(* IEC 61131-3 sources: IRIS-Project/LASAL CONTROL SOFTWARE/LasalProject_2025_09_25/Class/Motore_M4, 1 file *)

(* ---- Motore_M4.st ---- *)
(*!
<Class
	Name               = "Motore_M4"
	Revision           = "0.0"
	RealtimeTask       = "false"
	CyclicTask         = "true"
	DefCyclictime      = "100 ms"
	BackgroundTask     = "false"
	Sigmatek           = "false"
	OSInterface        = "false"
	HighPriority       = "false"
	Automatic          = "false"
	UpdateMode         = "Prescan"
	SharedCommandTable = "true"
	Objectsize         = "(720,180)">
	<Channels>
		<Server Name="ClassSvr" Visualized="false" Initialize="false" WriteProtected="true" Retentive="false"/>
		<Server Name="ErrorState" Visualized="false" Initialize="false" WriteProtected="true" Retentive="false"/>
		<Server Name="M4_Correction_Step" Visualized="false" Initialize="false" WriteProtected="false" Retentive="false"/>
		<Server Name="MotoreM4Step" Visualized="false" Initialize="false" WriteProtected="true" Retentive="false"/>
		<Server Name="s_1_3_pelletMode" Visualized="false" Initialize="false" WriteProtected="false" Retentive="false"/>
		<Server Name="s_calibrationMode" Visualized="false" Initialize="false" WriteProtected="false" Retentive="false"/>
		<Server Name="s_DischargeStatus" Visualized="false" Initialize="false" WriteProtected="false" Retentive="false"/>
		<Server Name="s_M4_Homed" Visualized="false" Initialize="false" WriteProtected="false" Retentive="false"/>
		<Server Name="s_measurement_ON" Visualized="false" Initialize="false" WriteProtected="true" Retentive="false"/>
		<Server Name="s_pelletInTrolley" Visualized="false" Initialize="false" WriteProtected="false" Retentive="false"/>
		<Server Name="s_pelletMeasured" Visualized="false" Initialize="false" WriteProtected="false" Retentive="false"/>
		<Server Name="s_target_misurati" Visualized="false" Initialize="false" WriteProtected="false" Retentive="false"/>
		<Client Name="c_MaxCurrent" Required="true" Internal="false"/>
		<Client Name="c_TimerDis" Required="false" Internal="false"/>
		<Client Name="c_TimerMov" Required="true" Internal="false"/>
		<Client Name="Comando_M4" Required="true" Internal="false"/>
		<Client Name="Comando_to_M8Class" Required="true" Internal="false"/>
		<Client Name="M4_LS" Required="false" Internal="false"/>
		<Client Name="SetPositionController" Required="true" Internal="false"/>
	</Channels>
</Class>
*)
Motore_M4 : CLASS
	TYPE
	  t_sequence_Cmd_motore_M4 :  //! <Type Public="true" Name="t_sequence_Cmd_motore_M4"/>
	  (
	    Cmd_motore_M4_idle,
	    Cmd_motore_M4_homing,
	    Cmd_motore_M4_phasing,
	    Cmd_motore_M4_movement,
	    Cmd_motore_M4_reset,
	    Cmd_motore_M4_stop,
	    Cmd_motore_M4_stopped,
	    Cmd_motore_M4_Error,
	    Cmd_motore_M4_movement_2
	  )$UDINT;
	END_TYPE
  //Servers:
	ClassSvr 	: SvrChCmd_DINT;
	MotoreM4Step 	: SvrCh_t_sequence_Cmd_motore_M4_PTofCls_Motore_M4;
	ErrorState 	: SvrCh__LMCAXIS_ERROR;
	s_measurement_ON 	: SvrCh_DINT;
	s_M4_Homed 	: SvrCh_DINT;
	M4_Correction_Step 	: SvrCh_DINT;
	s_target_misurati 	: SvrCh_DINT;
	s_calibrationMode 	: SvrCh_DINT;
	s_1_3_pelletMode 	: SvrCh_DINT;
	s_pelletMeasured 	: SvrCh_DINT;
	s_pelletInTrolley 	: SvrCh_DINT;
	s_DischargeStatus 	: SvrCh_DINT;
  //Clients:
	Comando_M4 	: CltChCmd__LMCAxis;
	Comando_to_M8Class 	: CltChCmd_Motore_M7;
	M4_LS 	: CltCh_DINT;
	c_MaxCurrent 	: CltCh_DINT;
	SetPositionController 	: CltCh_DINT;
	c_TimerDis 	: CltCh_DINT;
	c_TimerMov 	: CltCh_DINT;
  //Variables:
		ActCommand 	: t_sequence_Cmd_motore_M4;
		M4_homed 	: BOOL;
		M4_MovementStep 	: DINT;
		v_MeasurementStartOver 	: BOOL;
		v_DiscahrgeMisure_End 	: BOOL;
		v_M8_inBlockPos 	: BOOL;
		v_ErrorState 	: DINT;
		HomingStep 	: DINT;
		Movement_step 	: DINT;
		v_StartHomingCase 	: DINT;
		v_StartMovementCase 	: DINT;
		v_offset_Dis 	: DINT;
		v_target_misurati 	: DINT;
		v_M4_LS 	: DINT;
		v_ACK_M4_Mov 	: DINT;
		flag 	: DINT;
		v_startTimer 	: BOOL;
		v_pelletMeasured 	: DINT;
		v_pelletInTrolley 	: DINT;
		v_PelletAvailable 	: DINT;
  //Functions:

	FUNCTION VIRTUAL GLOBAL Init;

	FUNCTION VIRTUAL GLOBAL CyWork
		VAR_INPUT
			EAX 	: UDINT;
		END_VAR
		VAR_OUTPUT
			state (EAX) 	: UDINT;
		END_VAR;

	FUNCTION GLOBAL SetSequenceState
		VAR_INPUT
			Cmd_motore 	: t_sequence_Cmd_motore_M4;
			Motion_Type 	: DINT;
			StartCase 	: DINT;
		END_VAR
		VAR_OUTPUT
			retcode 	: DINT;
		END_VAR;

	FUNCTION GLOBAL GetHomedState
		VAR_OUTPUT
			Homed 	: BOOL;
		END_VAR;

	FUNCTION GLOBAL GetMisurationStartOver
		VAR_INPUT
			Status 	: BOOL;
		END_VAR;

	FUNCTION GLOBAL SetDischargeOver
		VAR_OUTPUT
			Status 	: BOOL;
		END_VAR;

	FUNCTION GLOBAL GetM8Status
		VAR_INPUT
			Status 	: BOOL;
		END_VAR
		VAR_OUTPUT
			retcode 	: DINT;
		END_VAR;

	FUNCTION GLOBAL GetErrorState
		VAR_OUTPUT
			ErrorState 	: DINT;
		END_VAR;

	FUNCTION GLOBAL GetMoveDone
		VAR_OUTPUT
			OutParam 	: DINT;
		END_VAR;

	FUNCTION GLOBAL GetPelletAvailable
		VAR_INPUT
			Param 	: DINT;
		END_VAR;
  //Tables:
	FUNCTION @STD
		VAR_OUTPUT
			ret_code	: CONFSTATES;
		END_VAR;
	FUNCTION GLOBAL TAB @CT_;
END_CLASS;

#pragma usingLtd _LMCAxis
#pragma usingLtd Motore_M7

FUNCTION VIRTUAL GLOBAL Motore_M4::CyWork
	VAR_INPUT
		EAX 	: UDINT;
	END_VAR
	VAR_OUTPUT
		state (EAX) 	: UDINT;
	END_VAR

  v_M4_LS:=M4_LS.Read();
  s_M4_Homed.Write(input:=M4_homed);

  s_target_misurati.Write(input:=v_target_misurati);

  case MotoreM4Step of
//===========================================================================================

    Cmd_motore_M4_idle:

    if Comando_M4.AxisError.HwError then
      v_ErrorState:=1;   ;
      MotoreM4Step:=Cmd_motore_M4_Error;
    end_if;
    v_ACK_M4_Mov:=0;
//===========================================================================================

    Cmd_motore_M4_homing:
    //lo muovo fino al click dello switch, questa posizione corrisponde a quella in cui un target, se nello slider, cade nella posizione di carico
    if Comando_M4.AxisError.HwError then
      v_ErrorState:=1;
      HomingStep:=0;
      MotoreM4Step:=Cmd_motore_M4_Error;
    end_if;

    case HomingStep of

    0://idle
      HomingStep:=v_StartHomingCase;

    5:
      if v_M4_LS then //Motore già in posizione.
        HomingStep:=50;
      else
        HomingStep:=10;
      end_if;

    10://POWER ON

      if (Comando_M4.AxisStatus.PowerOn=0) & (Comando_M4.AxisStatus.ReadyToPowerOn) then
        Comando_M4.PowerOn(Mode:=_LMCAXIS_MOVEDIRECTION::LMCAXIS_MOVE_ANY_WAY);
      elsif Comando_M4.AxisStatus.PowerOn then
        HomingStep:=20;
      end_if;

    20:

      Comando_M4.TuneAxis(Position:=P_M4_H, Speed:=V_M4, Accel:=A_M4, Mode:=LMCAXIS_TUNE_POSITON_IN_POSITIVE_DIRECTION, WaitTime:=0, Jerk:=J_M4);
      HomingStep:=30;

    30:
      if v_M4_LS=0 then //quando tocca LS
        Comando_M4.StopMove(Decel:=A_M4, Jerk:=J_M4);
        HomingStep:=40;
      end_if;

    40://Controllo che il motore si sia fermato

      if Comando_M4.AxisStatus.Standstill then
          Comando_M4.PowerOff(Mode:=LMCAXIS_IMMEDIATE_STOPP);
          HomingStep:=50;
      end_if;

    50:
       if Comando_M4.AxisStatus.PowerOn=0 then
          SetPositionController.Write(input:=0);
          M4_homed:=TRUE;
          MotoreM4Step:=Cmd_motore_M4_idle;
          v_StartHomingCase:=0;
       end_if;

    end_case;

//==================================================================================
     Cmd_motore_M4_movement:

    //
    //BLOCCO DI COMANDI PER MOVIMENTAZIONE MOTORE M4
    //
    //SI TROVA GIA' NELLA POSIZIONE IN CUI PUO' UN TARGET CADE

    if Comando_M4.AxisError.HwError then
      v_ErrorState:=1;
      Movement_step:=0;
      MotoreM4Step:=Cmd_motore_M4_Error;
    end_if;

    case Movement_step of

    0: //IDLE, ATTESA COMANDI| Il motore è già nella posizione di carica->tocca il LS
        Movement_step:=v_StartMovementCase;
    10://M2 si trova nella posizione corretta di caricamento DEVE RUOTARE NEL VERSO CORRETTO PER SCARICARE TARGET, compirà 1 giro completo (quasi)

     if (Comando_M4.AxisStatus.PowerOn=0) & (Comando_M4.AxisStatus.ReadyToPowerOn) then
        Comando_M4.PowerOn(Mode:=LMCAXIS_MOVE_ANY_WAY);
     elsif Comando_M4.AxisStatus.PowerOn then
        Movement_step:=20;
        s_DischargeStatus.Write(input:=0);
     end_if;

    20:

      if v_M8_inBlockPos then
        Movement_Step:=30;
      elsif v_M8_inBlockPos=FALSE then
        Comando_to_M8Class.SetSequenceState(Cmd_motore:=Motore_M7::Cmd_motore_M7_movement, Motion_type:=0, StartCase:=10);//dico al motore di andare in posizione di blocco
        Movement_Step:=25;
      end_if;

    25:
      if v_M8_inBlockPos=true then
        Movement_Step:=30;
        flag:=1;
      end_if;

    30:
      Comando_M4.MoveAbsolute(Position:=(P1_M4+v_offset_Dis), Speed:=V_M4, Accel:=A_M4, Decel:=A_M4, Jerk:=J_M4);
      Movement_Step:=40;

    40:
      IF Comando_M4.InPosition(Mode:=LMCAXIS_NO_POSITIONWINDOW, PositionWindow:=0) & Comando_M4.AxisStatus.Standstill  & v_MeasurementStartOver THEN //se ho scaricato target e dico che è pronto per la misurazione
      //FASE DI MISURAZIONE
        v_pelletMeasured+=1;
        s_pelletMeasured.Write(input:=v_pelletMeasured);
        c_TimerDis.Write(input:=1);
        c_TimerMov.Write(input:=0);
        s_measurement_ON.Write(input:=1);//MISURAZIONE ATTIVA
        s_DischargeStatus.Write(input:=1);
        v_target_misurati+=1;
        Movement_step:=50;
      END_IF;

    50:
      if v_MeasurementStartOver=FALSE then
        v_pelletMeasured+=1;
        s_pelletMeasured.Write(input:=v_pelletMeasured);
        c_TimerDis.Write(input:=0);
        Comando_to_M8Class.SetSequenceState(Cmd_motore:=Motore_M7::Cmd_motore_M7_movement, Motion_type:=1,StartCase:=10);//dico al motore di USCIRE dalla posizione di blocco
        v_target_misurati+=1;
        v_pelletInTrolley+=1;
        s_pelletInTrolley.Write(input:=v_pelletInTrolley);
        s_measurement_ON.Write(input:=0);
        v_offset_Dis+=1200000;

        if s_1_3_pelletMode.Read()=1 then
          Movement_Step:=80;
        elsif s_1_3_pelletMode.Read()=0 then
          Movement_Step:=60;
        end_if;

      end_if;

    60:
      if v_target_misurati<6 & Comando_to_M8Class.GetCoupledState()=FALSE then
        Movement_Step:=20;
      elsif v_target_misurati=6 & Comando_to_M8Class.GetCoupledState()=FALSE then
        Comando_M4.PowerOff(Mode:=LMCAXIS_IMMEDIATE_STOPP);
        Movement_Step:=70;
      end_if;

    70:
    if Comando_M4.AxisStatus.PowerOn=0 then
       s_DischargeStatus.Write(input:=2);
       v_DiscahrgeMisure_End:=TRUE;
       Movement_Step:=0;
       MotoreM4Step:=Cmd_motore_M4_idle;
    end_if;

    //Calibration Mode
    80:
      if Comando_to_M8Class.GetCoupledState()=FALSE & Comando_M4.AxisStatus.Standstill then
          Comando_M4.PowerOff(Mode:=LMCAXIS_IMMEDIATE_STOPP);
          Movement_Step:=70;
      end_if;

    end_case;
//========================================================================

    Cmd_motore_M4_movement_2:
    if Comando_M4.AxisError.HwError then
      v_ErrorState:=1;
      Movement_step:=0;
      MotoreM4Step:=Cmd_motore_M4_Error;
    end_if;

    case Movement_step of

    0: //IDLE, ATTESA COMANDI| Il motore è già nella posizione di carica->tocca il LS
        Movement_step:=v_StartMovementCase;
    10://M2 si trova nella posizione corretta di caricamento DEVE RUOTARE NEL VERSO CORRETTO PER SCARICARE TARGET, compirà 1 giro completo (quasi)

     if (Comando_M4.AxisStatus.PowerOn=0) & (Comando_M4.AxisStatus.ReadyToPowerOn) then
        Comando_M4.PowerOn(Mode:=LMCAXIS_MOVE_ANY_WAY);
     elsif Comando_M4.AxisStatus.PowerOn then
        Movement_step:=20;
     end_if;

    20:

      Comando_M4.MoveRelative(Position:=900000, Mode:=LMCAXIS_MOVE_RELATIVE_TO_POSITION , Speed:=V_M4, Accel:=A_M4, Decel:=A_M4, Jerk:=J_M4);
      Movement_step:=30;

    30:

      if Comando_M4.AxisStatus.InPosition then
        v_ACK_M4_Mov:=1;
        Movement_step:=40;
        Comando_M4.PowerOff(Mode:=LMCAXIS_IMMEDIATE_STOPP);
      end_if;

    40:
      Movement_Step:=0;
      v_StartMovementCase:=0;
      MotoreM4Step:=Cmd_motore_M4_idle;

    end_case;
//========================================================================

     Cmd_motore_M4_Error:

      ErrorState:=Comando_M4.AxisError; //AGGIORNAMENTO SERVER
      MotoreM4Step:=Cmd_motore_M4_stop;

//========================================================================
    Cmd_motore_M4_stop:

      if Comando_M4.AxisStatus.Standstill & Comando_M4.AxisStatus.PowerOn=0 then
        MotoreM4Step:=Cmd_motore_M4_stopped;
      else
        Comando_M4.QuickStop(Decel:=1000000);//se asse in errore non esegue neppure l'operazione perchè spento (e in errore)
        Comando_M4.PowerOff(Mode:=LMCAXIS_IMMEDIATE_STOPP);
      end_if;

//========================================================================
    Cmd_motore_M4_stopped:
    //ATTESA RESET

//========================================================================
    Cmd_motore_M4_reset:
      Comando_M4.QuitError();
      Comando_to_M8Class.SetSequenceState(Cmd_motore:=Motore_M7::Cmd_motore_M7_reset, Motion_type:=3, StartCase:=0);
      M4_homed:=FALSE;
      v_ErrorState:=0;
      if Comando_M4.AxisStatus.FiltRdy then
        MotoreM4Step:=Cmd_motore_M4_idle;
      end_if;

      v_MeasurementStartOver:=FALSE;
      v_DiscahrgeMisure_End:=FALSE;
      v_M8_inBlockPos:=0;
      v_offset_Dis:=0;
      v_target_misurati:=0;
      HomingStep:=0;
      Movement_step:=0;
      v_StartHomingCase:=0;
      v_StartMovementCase:=0;
      flag:=0;
      v_ACK_M4_Mov:=0;
      v_M4_LS:=0;
      v_ErrorState:=0;
      v_startTimer:=FALSE;
      s_calibrationMode.Write(input:=0);
      //s_1_3_pelletMode.Write(input:=0);
      s_DischargeStatus.Write(input:=0);

      if v_pelletMeasured/2>=v_PelletAvailable then
          v_pelletMeasured:=0;
          s_pelletMeasured.Write(input:=0);
          v_pelletInTrolley:=0;
          s_pelletInTrolley.Write(input:=0);
      end_if;

//========================================================================

  end_case;

	state := READY;
END_FUNCTION

FUNCTION GLOBAL Motore_M4::SetSequenceState
	VAR_INPUT
		Cmd_motore 	: t_sequence_Cmd_motore_M4;
		Motion_Type 	: DINT;
		StartCase 	: DINT;
	END_VAR
	VAR_OUTPUT
		retcode 	: DINT;
	END_VAR

  if Cmd_motore=Cmd_motore_M4_homing then
    v_StartHomingCase:=StartCase;
  elsif Cmd_motore=Cmd_motore_M4_movement then
    v_StartMovementCase:=StartCase;
  elsif Cmd_motore=Cmd_motore_M4_movement_2 then
    v_StartMovementCase:=StartCase;
  end_if;

  MotoreM4Step:=Cmd_motore;
  retcode:=true;
END_FUNCTION

FUNCTION VIRTUAL GLOBAL Motore_M4::Init
M4_homed:=FALSE;
v_MeasurementStartOver:=FALSE;
v_DiscahrgeMisure_End:=FALSE;
v_M8_inBlockPos:=0;

v_offset_Dis:=0;
v_target_misurati:=0;

HomingStep:=0;
Movement_step:=0;

v_StartHomingCase:=0;
v_StartMovementCase:=0;

flag:=0;

v_ACK_M4_Mov:=0;

v_M4_LS:=0;

v_ErrorState:=0;

v_startTimer:=FALSE;

v_pelletMeasured:=0;
v_pelletInTrolley:=0;

v_PelletAvailable:=0;

END_FUNCTION

FUNCTION GLOBAL Motore_M4::GetHomedState
	VAR_OUTPUT
		Homed 	: BOOL;
	END_VAR

  Homed:=M4_homed;
END_FUNCTION

FUNCTION GLOBAL Motore_M4::GetMisurationStartOver
	VAR_INPUT
		Status 	: BOOL;
	END_VAR
v_MeasurementStartOver:=Status;
END_FUNCTION

FUNCTION GLOBAL Motore_M4::SetDischargeOver
	VAR_OUTPUT
		Status 	: BOOL;
	END_VAR
Status:=v_DiscahrgeMisure_End;
END_FUNCTION

FUNCTION GLOBAL Motore_M4::GetM8Status
	VAR_INPUT
		Status 	: BOOL;
	END_VAR
	VAR_OUTPUT
		retcode 	: DINT;
	END_VAR

  v_M8_inBlockPos:=Status;
  retcode:=TRUE;

END_FUNCTION

FUNCTION GLOBAL Motore_M4::GetErrorState
	VAR_OUTPUT
		ErrorState 	: DINT;
	END_VAR
  ErrorState:=v_ErrorState;
END_FUNCTION

FUNCTION GLOBAL Motore_M4::GetMoveDone
	VAR_OUTPUT
		OutParam 	: DINT;
	END_VAR
OutParam:=v_ACK_M4_Mov;
END_FUNCTION

FUNCTION GLOBAL Motore_M4::GetPelletAvailable
	VAR_INPUT
		Param 	: DINT;
	END_VAR
v_PelletAvailable:=Param;
END_FUNCTION
